(* PLC project CoDeSys External Library Template, WAGO e!COCKPIT e!COCKPIT, author 3S - Smart Software Solutions GmbH *)
(* stored: creationDateTime 2019-10-29T12:37:19.7309586, version 3.5.5.30, modificationDateTime 2019-10-29T12:36:39.3744516, organization 3S - Smart Software Solutions GmbH *)
(* Library project template with all possible element types, docu and a sample project structure *)

FUNCTION_BLOCK fbPPPSZadajnikSR04P
  VAR_INPUT
    sKomunikat : alSTRINGKomunikat;  (* komunikat z systemu zewnętrznego *)
    intTablicaKomunikatowRozmiar : INT;  (* rozmiar tablicy danych wysyłkowych *)
    intModbusOdczytZapisZadanieRozmiar : INT;  (* rozmiar tablicy danych modbusa *)
    xTablicaKomunikatowHold : BOOL;  (* wstrzymanie komunikacji mniej ważnych komunikatów *)
    sIdInstancji : STRING;  (* parametr ID rolety np NS02L*202IBM**** *)
    sIdAplikacji : STRING;  (* parametr ID aplikacji np SO*******ECL*000 *)
    sMnemonik : STRING;  (* mnemonik właściciela - BCB* *)
    sMACAdres : STRING;  (* MAC adres sterownika *)
    sDaneZapasowe : STRING;  (* 6 znaków zapasu *)
    tCzasOpoznieniaRestartu : TIME;  (* czas opóźnienia po którym zaczynają być raportowane wartości *)
    sTypPomieszczenia : STRING;  (* typ pomieszczenia *)
    bAdres : BYTE;
    bKanalEnOcean : BYTE;
    sEnOceanID : STRING(10);
    tMinimalnyCzasRaportowania : TIME;
    tMaksymalnyCzasRaportowania : TIME;
    tCzasTimeoutEnOcean : TIME;
    xAutonomizacja : BOOL;
    xAutonomizacjaSztuczna : BOOL;
    xGlobalnaAutomatycznaKonfiguracja : BOOL;
    tCzestotliwoscAutomatycznejKonfiguracji : TIME;
    rRegulatorTemperaturyKp : REAL;
    rRegulatorTemperaturyTi : REAL;
    rRegulatorTemperaturyDeadZone : REAL;
    rTrybPracyAutonomizacja : REAL;  (* Domyślny tryb pracy *)
    rTemperaturaBazowaAutoAutonomizacja : REAL;  (* Domyślna wartość nastawy temperatury bazowej w trybie automatycznym *)
    rTemperaturaBazowaManAutonomizacja : REAL;  (* Domyślna wartość nastawy temperatury bazowej w trybie manualnym *)
    rSkalaPotencjometruAutonomizacja : REAL;  (* Domyślna skala potencjomentru *)
    rTemperaturaBazowaHMI : REAL := 293.15;  (* Temperatura bazowa z HMI *)
    intTrybPracyHMI : INT := 1;  (* 0 - ręczny; 1 - auto *)
    xPokazPanelHMI : BOOL := TRUE;  (* 0 - widoczny; 1 - niewidoczny *)
  END_VAR
  VAR_IN_OUT
    arModbusOdczytCykliczny : ARRAY[1..5000] OF typModbusOdczytCykliczny;
    arModbusStatusKomunikacji : ARRAY[1..256] OF INT;
    arModbusOdczytZapisZadanie : ARRAY[1..1000] OF typModbusOdczytZapisZadanie;
    intModbusOdczytZapisZadanieZnacznikZapisu : INT;
    arTablicaKomunikatow : alARRAYTablicaKomunikatow;
    intTablicaKomunikatowZnacznikZapisu : INT;
  END_VAR
  VAR_OUTPUT
    rWyjscieRgulatoraTemperatury : REAL;
    rDiagnostykaTemperaturaPomieszczenia : REAL;
    rDiagnostykaTemperaturaNastawiona : REAL;
    rDiagnostykaTemperaturaBazowa : REAL;
    rDiagnostykaKorektaTemperaturyPotencjometru : REAL;
    rDiagnostykaWyjscieRgulatoraTemperatury : REAL;
    intDiagnostykaTrybPracy : INT;
    sDiagnostykaEnOceanIDodczytany : STRING(10);
    wDiagnostykaCzasOdOstatniegoKomunikatu : WORD;
    rTemperaturaPomieszczenia : REAL;
  END_VAR
  VAR CONSTANT
    uintLiczbaRejestrowNaKanal : UINT := 20;
    uintPierwszyRejestr : UINT := 200;
    wEnOceanFunction : WORD := 16;
    wEnOceanType : WORD := 3;
    wEnOceanManufacturer : WORD := 2;
    intDomyslneHarmonogram : INT := enumPPPSHarmonogramy.Komfort;  (* domyślne nastawy po restarcie sterownika *)
    rDomyslneTemperaturaBazowaKomfort : REAL := 293.15;
    rDomyslneTemperaturaBazowaEkonomiczny : REAL := 292.15;
  END_VAR
  VAR
    uintFunctionModbusAdres : UINT;  (* definicja adresów rejestrów modbusowych *)
    uintTypeModbusAdres : UINT;
    uintManufacturerModbusAdres : UINT;
    uintEnOceanIDHiModbusAdres : UINT;
    uintEnOceanIDLoModbusAdres : UINT;
    uintCzasOdOstatniegoKomunikatuModbusAdres : UINT;
    uintPustyRejestr1ModbusAdres : UINT;
    uintStatusUrzadzeniaModbusAdres : UINT;
    uintPustyRejestr2ModbusAdres : UINT;
    uintTemperaturaPomieszczeniaOdczytanaModbusAdres : UINT;
    uintNastawaPotencjometruModbusAdres : UINT;
    xPierwszySkan : BOOL := TRUE;  (* uintLiczbaTelegramowModbusAdres : UINT; zmienne operacyjne *)
    intPetlaPierwszySkan : INT := 1;
    intRozkazTymczasowy : INT;
    arNastawyRegulatoraTemperatury : typConfigPIDController;
    fbRegulatorTemperatury : FbPIDController;
    intBlokadaWykonywaniaRozkazow : INT;
    intBlokadaWykonywaniaRozkazowZaraportowana : INT;
    intTrybPracy : INT;  (* Tryb pracy regulatora. *)
    intTrybPracyZaraportowana : INT;
    xTrybPracyZapisz : BOOL;  (* Trigger zapisu wartości w pamięci urządzenia. *)
    rTrybPracyZapis : REAL;  (* Wartość do zapisania w pamięci urządzenia. *)
    rTemperaturaBazowaAuto : REAL := 293.15;  (* Temperatura bazowa trybu automatycznego. *)
    rTemperaturaBazowaAutoZaraportowana : REAL;
    xTemperaturaBazowaAutoZapisz : BOOL;  (* Trigger zapisu wartości w pamięci urządzenia. *)
    rTemperaturaBazowaAutoZapis : REAL;  (* Wartość do zapisania w pamięci urządzenia. *)
    rTemperaturaBazowaMan : REAL := 293.15;  (* Temperatura bazowa trybu manualnego. *)
    rTemperaturaBazowaManZaraportowana : REAL;
    xTemperaturaBazowaManZapisz : BOOL;  (* Trigger zapisu wartości w pamięci urządzenia. *)
    rTemperaturaBazowaManZapis : REAL;  (* Wartość do zapisania w pamięci urządzenia. *)
    rSkalaPotencjometru : REAL;  (* Skala Potencjometru *)
    rSkalaPotencjometruZaraportowana : REAL;
    xSkalaPotencjometruZapisz : BOOL;  (* Trigger zapisu wartości w pamięci urządzenia. *)
    rSkalaPotencjometruZapis : REAL;  (* Wartość do zapisania w pamięci urządzenia. *)
    fbZadanieGrzania : fbFiltrWartoscAnalogowa;
    rZadanieGrzania : REAL;  (* Zadana grzania *)
    fbZadanieGrzaniaRaport : fbFiltrWartoscAnalogowa;
    rZadanieGrzaniaRaport : REAL;  (* Zadana grzania (raportowana) *)
    rZadanieGrzaniaRaportZaraportowana : REAL;
    rWartoscWejsciowaTemperaturyNastawionej : REAL;
    fbWyslanieKonfiguracji : TON;  (* definicja zmiennych i FB do odczytu wartości z modbusa *)
    xPozwolenieNaAutomatycznaKonfiguracje : BOOL;
    xResetTimerautomatycznejKonfiguracji : BOOL;
    wFunctionEnOceanOdczytana : WORD;
    wTypeEnOceanOdczytana : WORD;
    wManufacturerEnOceanOdczytana : WORD;
    sEnOceanIDodczytany : STRING(10);
    wEnOceanIDHi : WORD;
    wEnOceanIDLo : WORD;
    wEnOceanIDHiZapis : WORD;
    wEnOceanIDLoZapis : WORD;
    wCzasOdOstatniegoKomunikatu : WORD;
    fbTimeoutEnOcean : TON;
    wStatusUrzadzenia : WORD;
    wLiczbaTelegramow : WORD;
    uintLiczbaTelegramow : UINT;
    wPustyRejestr1 : WORD;  (* Rejestry odczytywane dla zgrupowania zapytania rejestrów Modbus *)
    wPustyRejestr2 : WORD;
    wTemperaturaPomieszczeniaOdczytana : WORD;
    fbTemperaturaPomieszczenia : fbFiltrWartoscAnalogowa;
    rTemperaturaPomieszczeniaZaraportowana : REAL;
    wNastawaPotencjometru : WORD;
    rTemperaturaNastawiona : REAL;
    rTemperaturaNastawionaZaraportowana : REAL;
    xPoInicjalizacji : BOOL := FALSE;  (* inicjalizacja *)
    fbInicjalizacyjnyTimer : TON;
    sDane : alSTRINGKomunikat;
    sWyslanyKomunikat : alSTRINGKomunikat;
    sKomunikatPamiec : alSTRINGKomunikat;
    sWyslanyKomunikatDummy : alSTRINGKomunikat;
    intPetla : INT;
    arErrorStan : ARRAY[0..3] OF INT;  (* tablica przechowująca statusy alarmowe *)
    arErrorKlasa : ARRAY[0..3] OF INT;  (* tablica przechowująca klasy danych alarmów *)
    sTempWartoscAtrybutu : STRING;
    rTempWartoscAtrybutu : REAL;
    intTempWartoscAtrybutu : INT;
    xRaport : BOOL;
    uintFunctionAdres : UINT;
    sPlakietkaHMI : STRING;  (* Plakietka pomieszczenia zawierająca numer piętra i pomieszczenia (na potrzeby webvisu) *)
    fnPrzywrocDomyslne : R_TRIG;  (* Przywracanie domyślnych wartości nastaw *)
    fbTaktowanieZapisywaniaModbus : TON;  (* Cykliczne żądanie zapisu danych do urządzenia *)
    xBrakKomunikacjiEnOcean : BOOL;  (* Brak komunikacji z urządzeniem po enOcean *)
    tonBrakKomunikacjiPLC : TON;
    xBrakKomunikacjiPLC : BOOL;
    xBrakKomunikacjiIZE : BOOL;
    rTemperaturaPomieszczeniaPamiec : REAL;  (* Temperatura zapamiętana w celu porównania z aktualną *)
    xBrakZmianyTemperatury : BOOL;  (* Flaga braku zmiany temperatury *)
    fbBrakZmianyTemperaturyTimer : TON;  (* Timer braku zmiany temperatury (24 godziny) *)
    xBladBrakZmianyTemperatury : BOOL;  (* Błąd braku zmiany temperatury *)
    xOsiagniecieTemperaturyZadanej : BOOL := FALSE;  (* Sprawdzanie czy została osiągnęta zadana temperatura *)
    xOsiagniecieTemperaturyZadanejZaraportowana : BOOL := FALSE;
    xFlagaTrybuPracy : BOOL := FALSE;
    rRoznicaTemperaturyZadanejOrazZaraportowanej : REAL;
  END_VAR

            (*			
Autor:					Paweł Kąkol, 2018-08-06, Artur Wyszomirski
Prawa majątkowe: 		Solwena Sp. z o.o., 
Aktualizacje:			
						2018-08-27-PK: dodanie algorytmu nadpisywania konfiguracji (uczenia) anteny
						2018-09-10-PK: dodanie regulatora temperatury oraz obsługi atrybutów potrzebnych do zadajnika z regulatorem, dodanie alarmowania Timeout komunikacji EnOcean
						2018-09-24-AWy: obsługa trybu manualnego i automatycznego
						2018-09-25-PK: dodanie domyślnego przyjmowania 21 st. C po restarcie sterownika, zanim nastąpi Autonomizacja i komunikacja z IZE.
						2018-15-10-AWy: obsługa harmonogramów
						2018-23-10-JB: przygotowanie atrybutów i alarmów do komunikacji z IZE
						2018-12-12-JB: napisanie od nowa obsługi ramek typu C i Q
						2019-02-26-JB: zmiana deadbandów w filtrach analogowych
						2019-04-08-AWy: usunięcie buga braku wysterowania grzejników w trybie manualnym (usunięcie intTrybPracy <> enumPPPSZadajnikTrybPracy.Manualny AND z linii 473)
						2019-05-13-AWy: zmiana wartości umieszczonej w atrybucie STERGRZ. Wartość rZadanieGrzania jest dzielona przez 100 tak, aby zakres STERGRZ mieścił się między 0 a 1.
						2019-05-16-AWy: modyfikacja warunku na raportowanie. Dopisane: AND arModbusStatusKomunikacji[bAdres] = enumModbusStatus.KomunikacjaPrawidlowa AND xPoInicjalizacji 
						2019-05-17-AWy: rozbicie zmiennej rTemperaturaBazowa na rTemperaturaBazowaAuto i rTemperaturaBazowaMan
						2019-05-21-AWy: modyfikacja przepisywania temperatury bazowej z IZE do lokalnej podczas regulacji IZE. 
						2019-06-05-AWy: załadowanie domyślnych trybów pracy i nastaw po przejściu w tryb autonomizacji
						2019-08-05-AWy: dodanie zmiennej sPlakietkaHMI.
						2019-08-14-AWy: zmiana fbPrzywrocDomyslne z przerzutnika RS na R_TRIG.
						2019-09-23-AWy: modyfikacja generowania wartości zmiennej xBrakKomunikacjiPLC
						2019-10-09-AWy: uzależnienie wystąpienia alarmu braku zmiany temperatury od stanu komunikacji 
						2019-10-10-AWy: przywrócenie zmiennej xBrakKomunikacjiEnOcean na potrzeby alarmów i webvisu z I etapu ENGIE
						2019-10-21-AWy: dodanie dodatkowego filtrowania zadanej grzania przy wysyłaniu ramek do IZE
						2019-10-22-AWy: usunięcie uintLiczbaTelegramowModbusAdres z odczytu po Modbusie
						
Opis:					fb służy do komunikacji po Modbus RTU za pośrednictwem bramek (STC65-RS485) EnOcean z zadajnikami FCP0 (SR04P) na budynkach PPP Sopot (ENGIE) 
*)

// Inicjalizacja sterownika
fbInicjalizacyjnyTimer(IN := NOT xPoInicjalizacji , PT := tCzasOpoznieniaRestartu);
IF fbInicjalizacyjnyTimer.Q THEN
	intTrybPracyZaraportowana := intTrybPracy;
	rTemperaturaBazowaAutoZaraportowana := rTemperaturaBazowaAuto;
	rTemperaturaBazowaManZaraportowana := rTemperaturaBazowaMan;
	rSkalaPotencjometruZaraportowana := rSkalaPotencjometru;
	rTemperaturaNastawionaZaraportowana := rTemperaturaNastawiona;
	rTemperaturaPomieszczeniaZaraportowana := rTemperaturaPomieszczenia;
	rZadanieGrzaniaRaportZaraportowana := rZadanieGrzaniaRaport;
	xOsiagniecieTemperaturyZadanej := xOsiagniecieTemperaturyZadanejZaraportowana;
	xPoInicjalizacji := TRUE;
END_IF

// Włącz autonomizację jeśli sterownik jest w stanie inicjalizacji lub nastąpiło wymuszenie autonomizacji
IF NOT xPoInicjalizacji OR xAutonomizacjaSztuczna = TRUE THEN
	xAutonomizacja := TRUE;
END_IF 

// Kontrola komunikacji
tonBrakKomunikacjiPLC(IN := (wCzasOdOstatniegoKomunikatu > 180 OR arModbusStatusKomunikacji[bAdres] <> enumModbusStatus.KomunikacjaPrawidlowa), PT := T#180S);
IF tonBrakKomunikacjiPLC.Q THEN
	xBrakKomunikacjiPLC := TRUE;
ELSE
	xBrakKomunikacjiPLC := FALSE;
END_IF

IF xAutonomizacja THEN
	xBrakKomunikacjiIZE := TRUE;
ELSE
	xBrakKomunikacjiIZE := FALSE;
END_IF

IF xPierwszySkan THEN
	xPierwszySkan := FALSE;
	WHILE arModbusOdczytCykliczny[intPetlaPierwszySkan].bAdresUrzadzenia <> 0 DO
		intPetlaPierwszySkan := intPetlaPierwszySkan + 1;
	END_WHILE
	
	//ustawienie parametrów regulatora temperatury
	arNastawyRegulatoraTemperatury.rKp := rRegulatorTemperaturyKp;
	arNastawyRegulatoraTemperatury.rTn := rRegulatorTemperaturyTi;
	arNastawyRegulatoraTemperatury.rTd := 0.0;
	arNastawyRegulatoraTemperatury.rOutputMax := 100.0;
	arNastawyRegulatoraTemperatury.rOutputMin := 0.0;
	arNastawyRegulatoraTemperatury.xPresetOn := TRUE;
	arNastawyRegulatoraTemperatury.rPresetValueOn := 0.0;
	arNastawyRegulatoraTemperatury.rPresetValueOff := 0.0;
	arNastawyRegulatoraTemperatury.rDeadZone := rRegulatorTemperaturyDeadZone;
	
	//wyznaczenie adresów rejestrów modbusowych
	uintFunctionModbusAdres := uintPierwszyRejestr + (uintLiczbaRejestrowNaKanal * (BYTE_TO_UINT(bKanalEnOcean) - 1));
	uintTypeModbusAdres := uintFunctionModbusAdres + 1;
	uintManufacturerModbusAdres := uintFunctionModbusAdres + 2;
	
	uintEnOceanIDHiModbusAdres := uintFunctionModbusAdres + 3;
	uintEnOceanIDLoModbusAdres := uintFunctionModbusAdres + 4;
	uintCzasOdOstatniegoKomunikatuModbusAdres := uintFunctionModbusAdres + 6;
	uintPustyRejestr1ModbusAdres := uintFunctionModbusAdres + 7;
	uintStatusUrzadzeniaModbusAdres := uintFunctionModbusAdres + 8;
	uintPustyRejestr2ModbusAdres := uintFunctionModbusAdres + 9;
	uintTemperaturaPomieszczeniaOdczytanaModbusAdres := uintFunctionModbusAdres + 10;
	uintNastawaPotencjometruModbusAdres := uintFunctionModbusAdres + 11;
	//uintLiczbaTelegramowModbusAdres := uintFunctionModbusAdres + 19;
	
//deklaracja rejestrow do odczytu
	//rejestry
	arModbusOdczytCykliczny[intPetlaPierwszySkan].bAdresUrzadzenia := bAdres;
	arModbusOdczytCykliczny[intPetlaPierwszySkan].bFunkcja := TO_BYTE(enumModbusKodyFunkcji.OdczytNRejestrow);
	arModbusOdczytCykliczny[intPetlaPierwszySkan].uiAdresRejestru := uintFunctionModbusAdres;
	arModbusOdczytCykliczny[intPetlaPierwszySkan].ltCzestotliwosc := TIME_TO_LTIME(tMaksymalnyCzasRaportowania);
	arModbusOdczytCykliczny[intPetlaPierwszySkan].pZmiennaReferencyjna := ADR(wFunctionEnOceanOdczytana);
	intPetlaPierwszySkan := intPetlaPierwszySkan + 1;
	
	arModbusOdczytCykliczny[intPetlaPierwszySkan].bAdresUrzadzenia := bAdres;
	arModbusOdczytCykliczny[intPetlaPierwszySkan].bFunkcja := TO_BYTE(enumModbusKodyFunkcji.OdczytNRejestrow);
	arModbusOdczytCykliczny[intPetlaPierwszySkan].uiAdresRejestru := uintTypeModbusAdres;
	arModbusOdczytCykliczny[intPetlaPierwszySkan].ltCzestotliwosc := TIME_TO_LTIME(tMaksymalnyCzasRaportowania);
	arModbusOdczytCykliczny[intPetlaPierwszySkan].pZmiennaReferencyjna := ADR(wTypeEnOceanOdczytana);
	intPetlaPierwszySkan := intPetlaPierwszySkan + 1;
	
	arModbusOdczytCykliczny[intPetlaPierwszySkan].bAdresUrzadzenia := bAdres;
	arModbusOdczytCykliczny[intPetlaPierwszySkan].bFunkcja := TO_BYTE(enumModbusKodyFunkcji.OdczytNRejestrow);
	arModbusOdczytCykliczny[intPetlaPierwszySkan].uiAdresRejestru := uintManufacturerModbusAdres;
	arModbusOdczytCykliczny[intPetlaPierwszySkan].ltCzestotliwosc := TIME_TO_LTIME(tMaksymalnyCzasRaportowania);
	arModbusOdczytCykliczny[intPetlaPierwszySkan].pZmiennaReferencyjna := ADR(wManufacturerEnOceanOdczytana);
	intPetlaPierwszySkan := intPetlaPierwszySkan + 1;
	
	arModbusOdczytCykliczny[intPetlaPierwszySkan].bAdresUrzadzenia := bAdres;
	arModbusOdczytCykliczny[intPetlaPierwszySkan].bFunkcja := TO_BYTE(enumModbusKodyFunkcji.OdczytNRejestrow);
	arModbusOdczytCykliczny[intPetlaPierwszySkan].uiAdresRejestru := uintEnOceanIDHiModbusAdres;
	arModbusOdczytCykliczny[intPetlaPierwszySkan].ltCzestotliwosc := TIME_TO_LTIME(tMaksymalnyCzasRaportowania);
	arModbusOdczytCykliczny[intPetlaPierwszySkan].pZmiennaReferencyjna := ADR(wEnOceanIDHi);
	intPetlaPierwszySkan := intPetlaPierwszySkan + 1;
	
	arModbusOdczytCykliczny[intPetlaPierwszySkan].bAdresUrzadzenia := bAdres;
	arModbusOdczytCykliczny[intPetlaPierwszySkan].bFunkcja := TO_BYTE(enumModbusKodyFunkcji.OdczytNRejestrow);
	arModbusOdczytCykliczny[intPetlaPierwszySkan].uiAdresRejestru := uintEnOceanIDLoModbusAdres;
	arModbusOdczytCykliczny[intPetlaPierwszySkan].ltCzestotliwosc := TIME_TO_LTIME(tMaksymalnyCzasRaportowania);
	arModbusOdczytCykliczny[intPetlaPierwszySkan].pZmiennaReferencyjna := ADR(wEnOceanIDLo);
	intPetlaPierwszySkan := intPetlaPierwszySkan + 1;
	
	arModbusOdczytCykliczny[intPetlaPierwszySkan].bAdresUrzadzenia := bAdres;
	arModbusOdczytCykliczny[intPetlaPierwszySkan].bFunkcja := TO_BYTE(enumModbusKodyFunkcji.OdczytNRejestrow);
	arModbusOdczytCykliczny[intPetlaPierwszySkan].uiAdresRejestru := uintCzasOdOstatniegoKomunikatuModbusAdres;
	arModbusOdczytCykliczny[intPetlaPierwszySkan].ltCzestotliwosc := TIME_TO_LTIME(tMinimalnyCzasRaportowania);
	arModbusOdczytCykliczny[intPetlaPierwszySkan].pZmiennaReferencyjna := ADR(wCzasOdOstatniegoKomunikatu);
	intPetlaPierwszySkan := intPetlaPierwszySkan + 1;
	
	arModbusOdczytCykliczny[intPetlaPierwszySkan].bAdresUrzadzenia := bAdres;
	arModbusOdczytCykliczny[intPetlaPierwszySkan].bFunkcja := TO_BYTE(enumModbusKodyFunkcji.OdczytNRejestrow);
	arModbusOdczytCykliczny[intPetlaPierwszySkan].uiAdresRejestru := uintPustyRejestr1ModbusAdres;
	arModbusOdczytCykliczny[intPetlaPierwszySkan].ltCzestotliwosc := TIME_TO_LTIME(tMinimalnyCzasRaportowania);
	arModbusOdczytCykliczny[intPetlaPierwszySkan].pZmiennaReferencyjna := ADR(wPustyRejestr1);
	intPetlaPierwszySkan := intPetlaPierwszySkan + 1;
	
	arModbusOdczytCykliczny[intPetlaPierwszySkan].bAdresUrzadzenia := bAdres;
	arModbusOdczytCykliczny[intPetlaPierwszySkan].bFunkcja := TO_BYTE(enumModbusKodyFunkcji.OdczytNRejestrow);
	arModbusOdczytCykliczny[intPetlaPierwszySkan].uiAdresRejestru := uintStatusUrzadzeniaModbusAdres;
	arModbusOdczytCykliczny[intPetlaPierwszySkan].ltCzestotliwosc := TIME_TO_LTIME(tMinimalnyCzasRaportowania);
	arModbusOdczytCykliczny[intPetlaPierwszySkan].pZmiennaReferencyjna := ADR(wStatusUrzadzenia);
	intPetlaPierwszySkan := intPetlaPierwszySkan + 1;
	
	arModbusOdczytCykliczny[intPetlaPierwszySkan].bAdresUrzadzenia := bAdres;
	arModbusOdczytCykliczny[intPetlaPierwszySkan].bFunkcja := TO_BYTE(enumModbusKodyFunkcji.OdczytNRejestrow);
	arModbusOdczytCykliczny[intPetlaPierwszySkan].uiAdresRejestru := uintPustyRejestr2ModbusAdres;
	arModbusOdczytCykliczny[intPetlaPierwszySkan].ltCzestotliwosc := TIME_TO_LTIME(tMinimalnyCzasRaportowania);
	arModbusOdczytCykliczny[intPetlaPierwszySkan].pZmiennaReferencyjna := ADR(wPustyRejestr2);
	intPetlaPierwszySkan := intPetlaPierwszySkan + 1;
	
	arModbusOdczytCykliczny[intPetlaPierwszySkan].bAdresUrzadzenia := bAdres;
	arModbusOdczytCykliczny[intPetlaPierwszySkan].bFunkcja := TO_BYTE(enumModbusKodyFunkcji.OdczytNRejestrow);
	arModbusOdczytCykliczny[intPetlaPierwszySkan].uiAdresRejestru := uintTemperaturaPomieszczeniaOdczytanaModbusAdres;
	arModbusOdczytCykliczny[intPetlaPierwszySkan].ltCzestotliwosc := TIME_TO_LTIME(tMinimalnyCzasRaportowania);
	arModbusOdczytCykliczny[intPetlaPierwszySkan].pZmiennaReferencyjna := ADR(wTemperaturaPomieszczeniaOdczytana);
	intPetlaPierwszySkan := intPetlaPierwszySkan + 1;	
	
	arModbusOdczytCykliczny[intPetlaPierwszySkan].bAdresUrzadzenia := bAdres;
	arModbusOdczytCykliczny[intPetlaPierwszySkan].bFunkcja := TO_BYTE(enumModbusKodyFunkcji.OdczytNRejestrow);
	arModbusOdczytCykliczny[intPetlaPierwszySkan].uiAdresRejestru := uintNastawaPotencjometruModbusAdres;
	arModbusOdczytCykliczny[intPetlaPierwszySkan].ltCzestotliwosc := TIME_TO_LTIME(tMinimalnyCzasRaportowania);
	arModbusOdczytCykliczny[intPetlaPierwszySkan].pZmiennaReferencyjna := ADR(wNastawaPotencjometru);
	intPetlaPierwszySkan := intPetlaPierwszySkan + 1;
(*	
	arModbusOdczytCykliczny[intPetlaPierwszySkan].bAdresUrzadzenia := bAdres;
	arModbusOdczytCykliczny[intPetlaPierwszySkan].bFunkcja := TO_BYTE(enumModbusKodyFunkcji.OdczytNRejestrow);
	arModbusOdczytCykliczny[intPetlaPierwszySkan].uiAdresRejestru := uintLiczbaTelegramowModbusAdres;
	arModbusOdczytCykliczny[intPetlaPierwszySkan].ltCzestotliwosc := TIME_TO_LTIME(tMinimalnyCzasRaportowania);
	arModbusOdczytCykliczny[intPetlaPierwszySkan].pZmiennaReferencyjna := ADR(wLiczbaTelegramow);
	intPetlaPierwszySkan := intPetlaPierwszySkan + 1;
*)	
(*	//przyjęcie nastaw domyślnych do momentu uzyskania nastaw z IZE lub przejścia w autonomizację
	IF intDomyslneHarmonogram = enumPPPSHarmonogramy.Ekonomiczny THEN
		rTemperaturaBazowaAuto := rDomyslneTemperaturaBazowaEkonomiczny;
	ELSE
		rTemperaturaBazowaAuto := rDomyslneTemperaturaBazowaKomfort;													
	END_IF
	intTrybPracy := enumPPPSZadajnikTrybPracy.Automatyczny;
	rSkalaPotencjometru := rSkalaPotencjometruAutonomizacja;	*)
END_IF

// Obsługa komunikatu przychodzacego z IZE
IF 	sKomunikat <> sKomunikatPamiec AND xPoInicjalizacji THEN
	sKomunikatPamiec := sKomunikat;
	IF fnIDOdbiorcyMatch(sKomunikat , sIdInstancji) THEN
		sDane := '';
		// Rozkaz typu C
		IF fnKomunikatTyp(sKomunikat) = 'C' AND NOT xAutonomizacja THEN
			// Blokada wykonywania rozkazów
			IF fnKomunikatDaneSzukajWartosci(sKomunikat,'BLOK=') = '0' THEN
				IF intBlokadaWykonywaniaRozkazow = 1 THEN
					intBlokadaWykonywaniaRozkazow := 0;
					xRaport := TRUE;
					ELSE	
					IF sDane <> '' THEN
					sDane := CONCAT(sDane , ';');
					END_IF
					sDane := CONCAT(sDane , 'BLOK=0');
				END_IF
			END_IF
			IF fnKomunikatDaneSzukajWartosci(sKomunikat,'BLOK=') = '1' THEN
				IF intBlokadaWykonywaniaRozkazow = 0 THEN
					intBlokadaWykonywaniaRozkazow := 1;
					xRaport := TRUE;
					ELSE
					IF sDane <> '' THEN
					sDane := CONCAT(sDane , ';');
					END_IF					
					sDane := CONCAT(sDane , 'BLOK=1');
				END_IF
			END_IF		

			IF intBlokadaWykonywaniaRozkazow = 0 THEN
				// Tryby pracy 
				fnKomunikatDaneZnajdzPorownajZapisz(sKomunikat := sKomunikat,
					sAtrybut := 'TRYB=',
					rAtrybutWartosc := rTrybPracyZapis,
					sDane := sDane,
					xAtrybutZapisz => xTrybPracyZapisz);	
				// Temperatura bazowa w trybie automatycznym
				fnKomunikatDaneZnajdzPorownajZapisz(sKomunikat := sKomunikat,
					sAtrybut := 'TEMPBAZAUTO=',
					rAtrybutWartosc := rTemperaturaBazowaAutoZapis,
					sDane := sDane,
					xAtrybutZapisz => xTemperaturaBazowaAutoZapisz);	
				// Temperatura bazowa w trybie manualnym
				fnKomunikatDaneZnajdzPorownajZapisz(sKomunikat := sKomunikat,
					sAtrybut := 'TEMPBAZMAN=',
					rAtrybutWartosc := rTemperaturaBazowaManZapis,
					sDane := sDane,
					xAtrybutZapisz => xTemperaturaBazowaManZapisz);
				// Skala potencjometru
				fnKomunikatDaneZnajdzPorownajZapisz(sKomunikat := sKomunikat,
					sAtrybut := 'SKALAPOT=',
					rAtrybutWartosc := rSkalaPotencjometruZapis,
					sDane := sDane,
					xAtrybutZapisz => xSkalaPotencjometruZapisz);
			END_IF
		END_IF	

		// Zapytanie typu Q
		IF fnKomunikatTyp(sKomunikat) = 'Q' AND arModbusStatusKomunikacji[bAdres] = enumModbusStatus.KomunikacjaPrawidlowa THEN
			IF fnKomunikatDaneSzukajWartosci(sKomunikat , 'BLOK=') = '?' OR fnKomunikatDaneSzukajWartosci(sKomunikat , 'ALL=') = '?' THEN
				fnKomunikatDaneDodaj(sDane := sDane , sAtrybut := 'BLOK=' , sWartosc := INT_TO_STRING(intBlokadaWykonywaniaRozkazow));	
			END_IF
			IF fnKomunikatDaneSzukajWartosci(sKomunikat , 'TRYB=') = '?' OR fnKomunikatDaneSzukajWartosci(sKomunikat , 'ALL=') = '?' THEN
				fnKomunikatDaneDodaj(sDane := sDane , sAtrybut := 'TRYB=' , sWartosc := INT_TO_STRING(intTrybPracy));	
			END_IF
			IF (fnKomunikatDaneSzukajWartosci(sKomunikat , 'TEMPBAZMAN=') = '?' OR fnKomunikatDaneSzukajWartosci(sKomunikat , 'ALL=') = '?') THEN
				fnKomunikatDaneDodaj(sDane := sDane , sAtrybut := 'TEMPBAZMAN=' , sWartosc := REAL_TO_STRING(rTemperaturaBazowaMan));	
			END_IF
			IF (fnKomunikatDaneSzukajWartosci(sKomunikat , 'TEMPBAZAUTO=') = '?' OR fnKomunikatDaneSzukajWartosci(sKomunikat , 'ALL=') = '?') THEN
				fnKomunikatDaneDodaj(sDane := sDane , sAtrybut := 'TEMPBAZAUTO=' , sWartosc := REAL_TO_STRING(rTemperaturaBazowaAuto));	
			END_IF
			IF fnKomunikatDaneSzukajWartosci(sKomunikat , 'SKALAPOT=') = '?' OR fnKomunikatDaneSzukajWartosci(sKomunikat , 'ALL=') = '?' THEN
				fnKomunikatDaneDodaj(sDane := sDane , sAtrybut := 'SKALAPOT=' , sWartosc := REAL_TO_STRING(rSkalaPotencjometru));	
			END_IF
			IF fnKomunikatDaneSzukajWartosci(sKomunikat , 'TEMP=') = '?' OR fnKomunikatDaneSzukajWartosci(sKomunikat , 'ALL=') = '?' THEN
				fnKomunikatDaneDodaj(sDane := sDane , sAtrybut := 'TEMP=' , sWartosc := REAL_TO_STRING(rTemperaturaPomieszczenia));	
			END_IF
			IF fnKomunikatDaneSzukajWartosci(sKomunikat , 'STERGRZ=') = '?' OR fnKomunikatDaneSzukajWartosci(sKomunikat , 'ALL=') = '?' THEN
				fnKomunikatDaneDodaj(sDane := sDane , sAtrybut := 'STERGRZ=' , sWartosc := REAL_TO_STRING(rZadanieGrzaniaRaport / 100));	
			END_IF
			IF fnKomunikatDaneSzukajWartosci(sKomunikat , 'TEMPNAS=') = '?' OR fnKomunikatDaneSzukajWartosci(sKomunikat , 'ALL=') = '?' THEN
				fnKomunikatDaneDodaj(sDane := sDane , sAtrybut := 'TEMPNAS=' , sWartosc := REAL_TO_STRING(rTemperaturaNastawiona));	
			END_IF
			IF fnKomunikatDaneSzukajWartosci(sKomunikat , 'DOGRZ=') = '?' OR fnKomunikatDaneSzukajWartosci(sKomunikat , 'ALL=') = '?' THEN
				fnKomunikatDaneDodaj(sDane := sDane , sAtrybut := 'DOGRZ=' , sWartosc := INT_TO_STRING(BOOL_TO_INT(xOsiagniecieTemperaturyZadanej)));	
			END_IF
			//pytanie o stany alarmów
			IF fnKomunikatDaneSzukajWartosci(sKomunikat , 'ALARM=') = '?' OR fnKomunikatDaneSzukajWartosci(sKomunikat , 'ALL=') = '?' THEN
				FOR intPetla := 1 TO 4 BY 1 DO
					//raportowanie typu E (stanów alarmów) na zapytanie typu Q
					IF arErrorStan[intPetla] <> enumAlarmWartosc.StanNieznany THEN
						fnZapiszKomunikat(	sCalyKomunikat := '' ,
											sTypKomunikatu := 'E' ,
											sMnemonik := sMnemonik ,
											sMACAdres := sMACAdres ,
											sIDNadawcy := sIdInstancji ,
											sIDOdbiorcy := sIdAplikacji ,
											sDaneZapasowe := sDaneZapasowe ,
											sDane := fnKomunikatDaneErrorRetry(xAktywny := arErrorStan[intPetla] = enumAlarmWartosc.StanAlarmowy , intKlasa := arErrorKlasa[intPetla] , intNumer := intPetla),
											arTablicaKomunikatow := arTablicaKomunikatow ,
											intTablicaKomunikatowZnacznikZapisu := intTablicaKomunikatowZnacznikZapisu ,
											intTablicaKomunikatowRozmiar := intTablicaKomunikatowRozmiar ,
											sWyslanyKomunikat := sWyslanyKomunikatDummy);
					END_IF
				END_FOR
			END_IF
		END_IF
		
		// Raportowanie typu A
		IF sDane <> '' THEN
			fnZapiszKomunikat(	sCalyKomunikat := '' ,
								sTypKomunikatu := 'A' ,
								sMnemonik := sMnemonik ,
								sMACAdres := sMACAdres ,
								sIDNadawcy := sIdInstancji ,
								sIDOdbiorcy := sIdAplikacji ,
								sDaneZapasowe := sDaneZapasowe ,
								sDane := sDane ,
								arTablicaKomunikatow := arTablicaKomunikatow ,
								intTablicaKomunikatowZnacznikZapisu := intTablicaKomunikatowZnacznikZapisu ,
								intTablicaKomunikatowRozmiar := intTablicaKomunikatowRozmiar ,
								sWyslanyKomunikat := sWyslanyKomunikatDummy);
		END_IF
	END_IF
END_IF

// Przywrócenie wartości domyślnych nastaw krzywej grzewczej i trybów pracy w przypadku restartu sterownika lub przejścia w stan autonomizacji (brak komunikacji z IZE)
fnPrzywrocDomyslne(CLK := xAutonomizacja);
IF fnPrzywrocDomyslne.Q THEN	
	IF intTrybPracy <> REAL_TO_INT(rTrybPracyAutonomizacja) THEN
		rTrybPracyZapis := rTrybPracyAutonomizacja;
		xTrybPracyZapisz := TRUE;
	END_IF
	IF rTemperaturaBazowaAuto <> rTemperaturaBazowaAutoAutonomizacja THEN
		rTemperaturaBazowaAutoZapis := rTemperaturaBazowaAutoAutonomizacja + 273.15;
		xTemperaturaBazowaAutoZapisz := TRUE;
	END_IF
	IF rTemperaturaBazowaMan <> rTemperaturaBazowaManAutonomizacja THEN
		rTemperaturaBazowaManZapis := rTemperaturaBazowaManAutonomizacja;
		xTemperaturaBazowaManZapisz := TRUE;
	END_IF
	IF rSkalaPotencjometru <> rSkalaPotencjometruAutonomizacja THEN
		rSkalaPotencjometruZapis := rSkalaPotencjometruAutonomizacja;
		xSkalaPotencjometruZapisz := TRUE;
	END_IF
END_IF	

// Zapisanie nastaw domyślnych lub otrzymanych w ramce C
IF xTrybPracyZapisz THEN
	intTrybPracy := REAL_TO_INT(rTrybPracyZapis);
	intTrybPracyHMI := REAL_TO_INT(rTrybPracyZapis);
	xTrybPracyZapisz := FALSE;
END_IF
IF xTemperaturaBazowaAutoZapisz THEN
	rTemperaturaBazowaAuto := rTemperaturaBazowaAutoZapis;
	xTemperaturaBazowaAutoZapisz := FALSE;
END_IF
IF xTemperaturaBazowaManZapisz THEN
	rTemperaturaBazowaMan := rTemperaturaBazowaManZapis;
	xTemperaturaBazowaManZapisz := FALSE;
END_IF
IF xSkalaPotencjometruZapisz THEN
	rSkalaPotencjometru := rSkalaPotencjometruZapis;
	xSkalaPotencjometruZapisz := FALSE;
END_IF

// Tryby pracy
IF xAutonomizacja THEN	// W trybie automonizacji pobieraj tryb pracy i temperaturę bazową z panelu WebVisu
	IF intTrybPracyHMI = enumPPPSZadajnikTrybPracy.Manualny THEN	
		intTrybPracy := enumPPPSZadajnikTrybPracy.Manualny;
		rTemperaturaBazowaMan := rTemperaturaBazowaHMI + 273.15;
	ELSE
		intTrybPracy := enumPPPSZadajnikTrybPracy.Automatyczny;
		rTemperaturaBazowaAuto := rTemperaturaBazowaAutoAutonomizacja + 273.15;
	END_IF
ELSE // W trybie sterowania z IZE pobieraj tryb pracy i temperaturę bazową z panelu WebVisu
	IF intTrybPracy = enumPPPSZadajnikTrybPracy.Manualny THEN
		intTrybPracyHMI := enumPPPSZadajnikTrybPracy.Manualny;
		rTemperaturaBazowaHMI := rTemperaturaBazowaMan - 273.15;
	ELSE
		intTrybPracyHMI := enumPPPSZadajnikTrybPracy.Automatyczny;
		rTemperaturaBazowaHMI := rTemperaturaBazowaAuto - 273.15;
	END_IF	
END_IF
						 
IF intTrybPracy = enumPPPSZadajnikTrybPracy.Manualny THEN 	
	rTemperaturaNastawiona := rTemperaturaBazowaMan; // W trybie manualnym nie uwzględniaj nastawy potencjometru na zadajniku
ELSE
	rTemperaturaNastawiona := ((WORD_TO_REAL(wNastawaPotencjometru) - 127.0) * rSkalaPotencjometru / 127.0) + rTemperaturaBazowaAuto; // W trybie automatycznym uwzględnij nastawę Potencjometru
END_IF

//Autokonfiguracja bramki EnOcean
sEnOceanIDodczytany := CONCAT(CONCAT(fnKonwersjaDEC_BYTE_TO_HEX_STRING(INT_TO_BYTE(WORD_TO_INT(wEnOceanIDHi / 256))), fnKonwersjaDEC_BYTE_TO_HEX_STRING(WORD_TO_BYTE(wEnOceanIDHi))), CONCAT(fnKonwersjaDEC_BYTE_TO_HEX_STRING(INT_TO_BYTE(WORD_TO_INT(wEnOceanIDLo / 256))), fnKonwersjaDEC_BYTE_TO_HEX_STRING(WORD_TO_BYTE(wEnOceanIDLo))));

fbWyslanieKonfiguracji(IN := ((xPozwolenieNaAutomatycznaKonfiguracje OR xGlobalnaAutomatycznaKonfiguracja) AND NOT xResetTimerautomatycznejKonfiguracji) , PT := tCzestotliwoscAutomatycznejKonfiguracji);
xResetTimerautomatycznejKonfiguracji := FALSE;

IF((xPozwolenieNaAutomatycznaKonfiguracje OR xGlobalnaAutomatycznaKonfiguracja) AND fbWyslanieKonfiguracji.Q) THEN
	//EnOcean ID urządzenia
	IF sEnOceanID <> sEnOceanIDodczytany THEN
		wEnOceanIDHiZapis := BYTE_TO_WORD(fnKonwersjaHEX_STRING_TO_DEC_BYTE(LEFT(sEnOceanID, 2))) * 256 + BYTE_TO_WORD(fnKonwersjaHEX_STRING_TO_DEC_BYTE(LEFT(RIGHT(sEnOceanID, 6), 2)));
		fnModbusZapisRejestru(	bAdresUrzadzenia := bAdres,
								bFunkcja := INT_TO_BYTE(enumModbusKodyFunkcji.ZapisRejestru),										
								uiAdresRejestru := uintEnOceanIDHiModbusAdres,
								pZmiennaReferencyjna := 0,
								wWartoscDoZapisania := wEnOceanIDHiZapis,
								intModbusOdczytZapisZadanieRozmiar := intModbusOdczytZapisZadanieRozmiar,
								arModbusOdczytZapisZadanie := arModbusOdczytZapisZadanie,
								intModbusOdczytZapisZadanieZnacznikZapisu := intModbusOdczytZapisZadanieZnacznikZapisu);
		wEnOceanIDLoZapis := BYTE_TO_WORD(fnKonwersjaHEX_STRING_TO_DEC_BYTE(LEFT(RIGHT(sEnOceanID, 4), 2))) * 256 + BYTE_TO_WORD(fnKonwersjaHEX_STRING_TO_DEC_BYTE(RIGHT(sEnOceanID, 2)));
		fnModbusZapisRejestru(	bAdresUrzadzenia := bAdres,
								bFunkcja := INT_TO_BYTE(enumModbusKodyFunkcji.ZapisRejestru),										
								uiAdresRejestru := uintEnOceanIDLoModbusAdres,
								pZmiennaReferencyjna := 0,
								wWartoscDoZapisania := wEnOceanIDLoZapis,
								intModbusOdczytZapisZadanieRozmiar := intModbusOdczytZapisZadanieRozmiar,
								arModbusOdczytZapisZadanie := arModbusOdczytZapisZadanie,
								intModbusOdczytZapisZadanieZnacznikZapisu := intModbusOdczytZapisZadanieZnacznikZapisu);
	END_IF
	//stałe wartości dla danego typu urządzeń
	IF wFunctionEnOceanOdczytana <> wEnOceanFunction THEN
		fnModbusZapisRejestru(	bAdresUrzadzenia := bAdres,
								bFunkcja := INT_TO_BYTE(enumModbusKodyFunkcji.ZapisRejestru),										
								uiAdresRejestru := uintFunctionModbusAdres,
								pZmiennaReferencyjna := 0,
								wWartoscDoZapisania := wEnOceanFunction,
								intModbusOdczytZapisZadanieRozmiar := intModbusOdczytZapisZadanieRozmiar,
								arModbusOdczytZapisZadanie := arModbusOdczytZapisZadanie,
								intModbusOdczytZapisZadanieZnacznikZapisu := intModbusOdczytZapisZadanieZnacznikZapisu);
	END_IF
	IF wTypeEnOceanOdczytana <> wEnOceanType THEN
		fnModbusZapisRejestru(	bAdresUrzadzenia := bAdres,
								bFunkcja := INT_TO_BYTE(enumModbusKodyFunkcji.ZapisRejestru),										
								uiAdresRejestru := uintTypeModbusAdres,
								pZmiennaReferencyjna := 0,
								wWartoscDoZapisania := wEnOceanType,
								intModbusOdczytZapisZadanieRozmiar := intModbusOdczytZapisZadanieRozmiar,
								arModbusOdczytZapisZadanie := arModbusOdczytZapisZadanie,
								intModbusOdczytZapisZadanieZnacznikZapisu := intModbusOdczytZapisZadanieZnacznikZapisu);
	END_IF
	IF wManufacturerEnOceanOdczytana <> wEnOceanManufacturer THEN
		fnModbusZapisRejestru(	bAdresUrzadzenia := bAdres,
								bFunkcja := INT_TO_BYTE(enumModbusKodyFunkcji.ZapisRejestru),										
								uiAdresRejestru := uintManufacturerModbusAdres,
								pZmiennaReferencyjna := 0,
								wWartoscDoZapisania := wEnOceanManufacturer,
								intModbusOdczytZapisZadanieRozmiar := intModbusOdczytZapisZadanieRozmiar,
								arModbusOdczytZapisZadanie := arModbusOdczytZapisZadanie,
								intModbusOdczytZapisZadanieZnacznikZapisu := intModbusOdczytZapisZadanieZnacznikZapisu);
	END_IF
	xResetTimerautomatycznejKonfiguracji := TRUE;
END_IF

//sprawdzanie Timeout komunikacji
fbTimeoutEnOcean(IN := ((wCzasOdOstatniegoKomunikatu > 120) AND arModbusStatusKomunikacji[bAdres] = enumModbusStatus.KomunikacjaPrawidlowa) , PT := tCzasTimeoutEnOcean);	
							
fbTemperaturaPomieszczenia(	rWartoscWejsciowa := WORD_TO_REAL(wTemperaturaPomieszczeniaOdczytana),
							rDeadband := 0.1,
							tCzasMinimalny := tMinimalnyCzasRaportowania,
							tCzasMaksymalny := tMaksymalnyCzasRaportowania,
							rWynikMnoznik := (-40.0 / 255.0),
							rWynikOffset := 273.15 + 40.0,
							rWartoscWejsciowaZaraportowana := rTemperaturaPomieszczeniaZaraportowana,
							rWartoscWyjsciowa => rTemperaturaPomieszczenia);

//regulator PI
fbRegulatorTemperatury( xEnable := TRUE,
	rReferenceValue := rTemperaturaNastawiona,
	rActualValue := rTemperaturaPomieszczenia,
	typConfigParameters := arNastawyRegulatoraTemperatury,
	rY => rWyjscieRgulatoraTemperatury);

fbZadanieGrzania(rWartoscWejsciowa := rWyjscieRgulatoraTemperatury,
	rDeadband := 0.25,
	tCzasMinimalny := tMinimalnyCzasRaportowania,
	tCzasMaksymalny := tMaksymalnyCzasRaportowania,
	rWynikMnoznik := 1,
	rWynikOffset := 0.0,
	rWartoscWejsciowaZaraportowana := rZadanieGrzania,
	rWartoscWyjsciowa => rZadanieGrzania);		
	
// Raportowanie zadanej grzania
fbZadanieGrzaniaRaport(rWartoscWejsciowa := rZadanieGrzania,
	rDeadband := 10,
	tCzasMinimalny := tMinimalnyCzasRaportowania,
	tCzasMaksymalny := tMaksymalnyCzasRaportowania,
	rWynikMnoznik := 1,
	rWynikOffset := 0.0,
	rWartoscWejsciowaZaraportowana := rZadanieGrzaniaRaportZaraportowana,
	rWartoscWyjsciowa => rZadanieGrzaniaRaport);		
	
// Nowy filtr "antypyćkowy"
IF rZadanieGrzania < 0.25 THEN
	rZadanieGrzania := 0;
	rZadanieGrzaniaRaport := 0;
ELSIF rZadanieGrzania > 99.75 THEN
	rZadanieGrzania := 100;
	rZadanieGrzaniaRaport := 100;	
END_IF
(*
// FILTR ANTY_PYĆKOWY
rRoznicaTemperaturyZadanejOrazZaraportowanej := rZadanieGrzania - rZadanieGrzaniaZaraportowana;
IF rRoznicaTemperaturyZadanejOrazZaraportowanej < 0.25 AND rRoznicaTemperaturyZadanejOrazZaraportowanej > 0 AND rZadanieGrzania < 1.0 THEN
	rZadanieGrzania := rZadanieGrzaniaZaraportowana;
END_IF	

IF rRoznicaTemperaturyZadanejOrazZaraportowanej > - 0.25 AND rRoznicaTemperaturyZadanejOrazZaraportowanej < 0 AND rZadanieGrzania > 99.0 THEN
	rZadanieGrzania := rZadanieGrzaniaZaraportowana;
END_IF	
	*)		
///////Diagnostyka na czas uruchomień////////
	rDiagnostykaTemperaturaPomieszczenia := rTemperaturaPomieszczenia;
	rDiagnostykaTemperaturaNastawiona := rTemperaturaNastawiona;
	rDiagnostykaTemperaturaBazowa := rTemperaturaBazowaAuto;
	rDiagnostykaKorektaTemperaturyPotencjometru := (WORD_TO_REAL(wNastawaPotencjometru) - 127.0) * rSkalaPotencjometru / 127.0;
	rDiagnostykaWyjscieRgulatoraTemperatury := rWyjscieRgulatoraTemperatury;
	intDiagnostykaTrybPracy := intTrybPracy;
	sDiagnostykaEnOceanIDodczytany := sEnOceanIDodczytany;
	wDiagnostykaCzasOdOstatniegoKomunikatu := wCzasOdOstatniegoKomunikatu;
//////////////////////////////////////////////		
IF (intBlokadaWykonywaniaRozkazow <> intBlokadaWykonywaniaRozkazowZaraportowana OR intTrybPracy <> intTrybPracyZaraportowana OR rTemperaturaBazowaAuto <> rTemperaturaBazowaAutoZaraportowana OR 
	rSkalaPotencjometru <> rSkalaPotencjometruZaraportowana OR rTemperaturaNastawiona <> rTemperaturaNastawionaZaraportowana OR rTemperaturaPomieszczenia <> rTemperaturaPomieszczeniaZaraportowana OR 
	rZadanieGrzaniaRaport <> rZadanieGrzaniaRaportZaraportowana OR xOsiagniecieTemperaturyZadanej <> xOsiagniecieTemperaturyZadanejZaraportowana OR rTemperaturaBazowaMan <> rTemperaturaBazowaManZaraportowana) AND 
	arModbusStatusKomunikacji[bAdres] = enumModbusStatus.KomunikacjaPrawidlowa AND xPoInicjalizacji THEN
	xRaport := TRUE;
END_IF

IF xRaport THEN
	sDane := '';
	xRaport := FALSE;
	IF intBlokadaWykonywaniaRozkazow <> intBlokadaWykonywaniaRozkazowZaraportowana THEN
		intBlokadaWykonywaniaRozkazowZaraportowana := intBlokadaWykonywaniaRozkazow;
		fnKomunikatDaneDodaj(sDane := sDane , sAtrybut := 'BLOK=' , sWartosc := INT_TO_STRING(intBlokadaWykonywaniaRozkazow));	
	END_IF
	IF intTrybPracy <> intTrybPracyZaraportowana THEN
		intTrybPracyZaraportowana := intTrybPracy;
		fnKomunikatDaneDodaj(sDane := sDane , sAtrybut := 'TRYB=' , sWartosc := INT_TO_STRING(intTrybPracy));	
	END_IF
	IF (rTemperaturaBazowaMan <> rTemperaturaBazowaManZaraportowana) THEN
		rTemperaturaBazowaManZaraportowana := rTemperaturaBazowaMan;
		fnKomunikatDaneDodaj(sDane := sDane , sAtrybut := 'TEMPBAZMAN=' , sWartosc := REAL_TO_STRING(rTemperaturaBazowaMan));	
	END_IF
	IF (rTemperaturaBazowaAuto <> rTemperaturaBazowaAutoZaraportowana) THEN
		rTemperaturaBazowaAutoZaraportowana := rTemperaturaBazowaAuto;
		fnKomunikatDaneDodaj(sDane := sDane , sAtrybut := 'TEMPBAZAUTO=' , sWartosc := REAL_TO_STRING(rTemperaturaBazowaAuto));	
	END_IF
	IF rSkalaPotencjometru <> rSkalaPotencjometruZaraportowana THEN
		rSkalaPotencjometruZaraportowana := rSkalaPotencjometru;
		fnKomunikatDaneDodaj(sDane := sDane , sAtrybut := 'SKALAPOT=' , sWartosc := REAL_TO_STRING(rSkalaPotencjometru));	
	END_IF
	IF rTemperaturaNastawiona <> rTemperaturaNastawionaZaraportowana THEN
		rTemperaturaNastawionaZaraportowana := rTemperaturaNastawiona;
		fnKomunikatDaneDodaj(sDane := sDane , sAtrybut := 'TEMPNAS=' , sWartosc := REAL_TO_STRING(rTemperaturaNastawiona));	
	END_IF
	IF rTemperaturaPomieszczenia <> rTemperaturaPomieszczeniaZaraportowana THEN
		rTemperaturaPomieszczeniaZaraportowana := rTemperaturaPomieszczenia;
		fnKomunikatDaneDodaj(sDane := sDane , sAtrybut := 'TEMP=' , sWartosc := REAL_TO_STRING(rTemperaturaPomieszczenia));	
	END_IF
	IF rZadanieGrzaniaRaport <> rZadanieGrzaniaRaportZaraportowana THEN
		rZadanieGrzaniaRaportZaraportowana := rZadanieGrzaniaRaport;	
		fnKomunikatDaneDodaj(sDane := sDane , sAtrybut := 'STERGRZ=' , sWartosc := REAL_TO_STRING(rZadanieGrzaniaRaport / 100));	
	END_IF
	IF xOsiagniecieTemperaturyZadanej <> xOsiagniecieTemperaturyZadanejZaraportowana THEN
		xOsiagniecieTemperaturyZadanejZaraportowana := xOsiagniecieTemperaturyZadanej;
		fnKomunikatDaneDodaj(sDane := sDane , sAtrybut := 'DOGRZ=' , sWartosc := INT_TO_STRING(BOOL_TO_INT(xOsiagniecieTemperaturyZadanej)));	
	END_IF
	
(*	IF rTemperaturaPomieszczeniaMIN <> rTemperaturaPomieszczeniaMINZaraportowana OR rTemperaturaPomieszczeniaMAX <> rTemperaturaPomieszczeniaMAXZaraportowana THEN
		
		fnKomunikatDaneDodaj(sDane := sDane , sAtrybut := 'TEMPPOC=' , sWartosc := REAL_TO_STRING(rTemperaturaPomieszczeniaPOCZATKOWA));
		rTemperaturaPomieszczeniaPOCZATKOWA := rTemperaturaPomieszczenia;
		
		rTemperaturaPomieszczeniaKONCOWA := rTemperaturaPomieszczenia;
		fnKomunikatDaneDodaj(sDane := sDane , sAtrybut := 'TEMPKON=' , sWartosc := REAL_TO_STRING(rTemperaturaPomieszczeniaKONCOWA));
		
		rTemperaturaPomieszczeniaMINZaraportowana := rTemperaturaPomieszczeniaMIN;
		fnKomunikatDaneDodaj(sDane := sDane , sAtrybut := 'TEMPMIN=' , sWartosc := REAL_TO_STRING(rTemperaturaPomieszczeniaMIN));
		rZmiennaProcesowaMinimumTemperatury := 500.0;
		
		rTemperaturaPomieszczeniaMAXZaraportowana := rTemperaturaPomieszczeniaMAX;
		fnKomunikatDaneDodaj(sDane := sDane , sAtrybut := 'TEMPMAX=' , sWartosc := REAL_TO_STRING(rTemperaturaPomieszczeniaMAX));
		rZmiennaProcesowaMaximumTemperatury := -1.0;
		
		fnKomunikatDaneDodaj(sDane := sDane , sAtrybut := 'TEMPSRE=' , sWartosc := REAL_TO_STRING(rTemperaturaPomieszczeniaSREDNIA));
		rTemperaturaPomieszczeniaSREDNIA := 0.0;
		
		fnKomunikatDaneDodaj(sDane := sDane , sAtrybut := 'TEMPMED=' , sWartosc := REAL_TO_STRING(rTemperaturaPomieszczeniaMEDIANA));
		rTemperaturaPomieszczeniaMEDIANA := -1.0;
	END_IF
*)

	IF sDane <> '' AND xPoInicjalizacji THEN
		fnZapiszKomunikat(	sCalyKomunikat := '' ,
							sTypKomunikatu := 'M' ,
							sMnemonik := sMnemonik ,
							sMACAdres := sMACAdres ,
							sIDNadawcy := sIdInstancji ,
							sIDOdbiorcy := sIdAplikacji ,
							sDaneZapasowe := sDaneZapasowe ,
							sDane := sDane ,
							arTablicaKomunikatow := arTablicaKomunikatow ,
							intTablicaKomunikatowZnacznikZapisu := intTablicaKomunikatowZnacznikZapisu ,
							intTablicaKomunikatowRozmiar := intTablicaKomunikatowRozmiar ,
							sWyslanyKomunikat := sWyslanyKomunikat);
	END_IF
END_IF

// Sprawdzanie czy pomiar temperatury działa (odczyt jest niepoprawny, jeśli nie zmienił wartości w przeciągu doby)
IF rTemperaturaPomieszczeniaPamiec = rTemperaturaPomieszczenia THEN
	xBrakZmianyTemperatury := TRUE;
ELSE
	xBrakZmianyTemperatury := FALSE;	
END_IF
fbBrakZmianyTemperaturyTimer(IN := xBrakZmianyTemperatury, PT := T#12H);
rTemperaturaPomieszczeniaPamiec := rTemperaturaPomieszczenia;
IF fbBrakZmianyTemperaturyTimer.Q AND NOT xBrakKomunikacjiPLC THEN
	xBladBrakZmianyTemperatury := TRUE;
ELSE
	xBladBrakZmianyTemperatury := FALSE;
END_IF

// Sprawdzanie czy została osiągnęta zadana temperatura
IF rTemperaturaPomieszczenia >= rTemperaturaNastawiona THEN
	xOsiagniecieTemperaturyZadanej  := TRUE;
END_IF
IF rTemperaturaPomieszczenia <= rTemperaturaNastawiona - 0.4 THEN
	xOsiagniecieTemperaturyZadanej := FALSE;	
END_IF

// obsługa alarmów do zadajnika
	//brak komunikacji po EnOcean
IF arErrorStan[enumPPPSZadajnikError.BrakKomunikacji] <> enumAlarmWartosc.StanAlarmowy AND fbTimeoutEnOcean.Q AND arModbusStatusKomunikacji[bAdres] = enumModbusStatus.KomunikacjaPrawidlowa THEN
	arErrorStan[enumPPPSZadajnikError.BrakKomunikacji] := enumAlarmWartosc.StanAlarmowy;
	xBrakKomunikacjiEnOcean := TRUE;
	arErrorKlasa[enumPPPSZadajnikError.BrakKomunikacji] := enumPPPSZadajnikErrorKlasa.BrakKomunikacji;
	IF xPoInicjalizacji THEN
		fnZapiszKomunikat(	sCalyKomunikat := '' ,
							sTypKomunikatu := 'E' ,
							sMnemonik := sMnemonik ,
							sMACAdres := sMACAdres ,
							sIDNadawcy := sIdInstancji ,
							sIDOdbiorcy := sIdAplikacji ,
							sDaneZapasowe := sDaneZapasowe ,
							sDane := fnKomunikatDaneError(xAktywny := TRUE , intKlasa := enumPPPSZadajnikErrorKlasa.BrakKomunikacji , intNumer := enumPPPSZadajnikError.BrakKomunikacji),
							arTablicaKomunikatow := arTablicaKomunikatow ,
							intTablicaKomunikatowZnacznikZapisu := intTablicaKomunikatowZnacznikZapisu ,
							intTablicaKomunikatowRozmiar := intTablicaKomunikatowRozmiar ,
							sWyslanyKomunikat := sWyslanyKomunikatDummy);
	END_IF
END_IF
IF arErrorStan[enumPPPSZadajnikError.BrakKomunikacji] <> enumAlarmWartosc.StanNormalny AND NOT fbTimeoutEnOcean.Q AND arModbusStatusKomunikacji[bAdres] = enumModbusStatus.KomunikacjaPrawidlowa THEN
	arErrorStan[enumPPPSZadajnikError.BrakKomunikacji] := enumAlarmWartosc.StanNormalny;
	xBrakKomunikacjiEnOcean := FALSE;
	arErrorKlasa[enumPPPSZadajnikError.BrakKomunikacji] := enumPPPSZadajnikErrorKlasa.BrakKomunikacji;
	IF xPoInicjalizacji THEN
		fnZapiszKomunikat(	sCalyKomunikat := '' ,
							sTypKomunikatu := 'E' ,
							sMnemonik := sMnemonik ,
							sMACAdres := sMACAdres ,
							sIDNadawcy := sIdInstancji ,
							sIDOdbiorcy := sIdAplikacji ,
							sDaneZapasowe := sDaneZapasowe ,
							sDane := fnKomunikatDaneError(xAktywny := FALSE , intKlasa := enumPPPSZadajnikErrorKlasa.BrakKomunikacji , intNumer := enumPPPSZadajnikError.BrakKomunikacji),
							arTablicaKomunikatow := arTablicaKomunikatow ,
							intTablicaKomunikatowZnacznikZapisu := intTablicaKomunikatowZnacznikZapisu ,
							intTablicaKomunikatowRozmiar := intTablicaKomunikatowRozmiar ,
							sWyslanyKomunikat := sWyslanyKomunikatDummy);
	END_IF
END_IF
// Alarm czujnika temperatury
IF arErrorStan[enumPPPSZadajnikError.AlarmCzujnika] <> enumAlarmWartosc.StanAlarmowy AND xBladBrakZmianyTemperatury AND arModbusStatusKomunikacji[bAdres] = enumModbusStatus.KomunikacjaPrawidlowa THEN
	arErrorStan[enumPPPSZadajnikError.AlarmCzujnika] := enumAlarmWartosc.StanAlarmowy;
	arErrorKlasa[enumPPPSZadajnikError.AlarmCzujnika] := enumPPPSZadajnikErrorKlasa.AlarmCzujnika;
	IF xPoInicjalizacji THEN
		fnZapiszKomunikat(	sCalyKomunikat := '' ,
							sTypKomunikatu := 'E' ,
							sMnemonik := sMnemonik ,
							sMACAdres := sMACAdres ,
							sIDNadawcy := sIdInstancji ,
							sIDOdbiorcy := sIdAplikacji ,
							sDaneZapasowe := sDaneZapasowe ,
							sDane := fnKomunikatDaneError(xAktywny := TRUE , intKlasa := enumPPPSZadajnikErrorKlasa.AlarmCzujnika , intNumer := enumPPPSZadajnikError.AlarmCzujnika),
							arTablicaKomunikatow := arTablicaKomunikatow ,
							intTablicaKomunikatowZnacznikZapisu := intTablicaKomunikatowZnacznikZapisu ,
							intTablicaKomunikatowRozmiar := intTablicaKomunikatowRozmiar ,
							sWyslanyKomunikat := sWyslanyKomunikatDummy);
	END_IF
END_IF

IF arErrorStan[enumPPPSZadajnikError.AlarmCzujnika] <> enumAlarmWartosc.StanNormalny AND NOT xBladBrakZmianyTemperatury AND arModbusStatusKomunikacji[bAdres] = enumModbusStatus.KomunikacjaPrawidlowa THEN
	arErrorStan[enumPPPSZadajnikError.AlarmCzujnika] := enumAlarmWartosc.StanNormalny;
	arErrorKlasa[enumPPPSZadajnikError.AlarmCzujnika] := enumPPPSZadajnikErrorKlasa.AlarmCzujnika;
	IF xPoInicjalizacji THEN
		fnZapiszKomunikat(	sCalyKomunikat := '' ,
							sTypKomunikatu := 'E' ,
							sMnemonik := sMnemonik ,
							sMACAdres := sMACAdres ,
							sIDNadawcy := sIdInstancji ,
							sIDOdbiorcy := sIdAplikacji ,
							sDaneZapasowe := sDaneZapasowe ,
							sDane := fnKomunikatDaneError(xAktywny := FALSE , intKlasa := enumPPPSZadajnikErrorKlasa.AlarmCzujnika , intNumer := enumPPPSZadajnikError.AlarmCzujnika),
							arTablicaKomunikatow := arTablicaKomunikatow ,
							intTablicaKomunikatowZnacznikZapisu := intTablicaKomunikatowZnacznikZapisu ,
							intTablicaKomunikatowRozmiar := intTablicaKomunikatowRozmiar ,
							sWyslanyKomunikat := sWyslanyKomunikatDummy);
	END_IF
END_IF

// Plakietka pomieszczenia (numer piętra.numer pomieszczenia)
sPlakietkaHMI := CONCAT(STR1 := MID(sIdInstancji, LEN := 2, POS := 3), '.');
sPlakietkaHMI := CONCAT(sPlakietkaHMI, MID(STR := sIdInstancji, LEN := 3, POS := 7));
          
END_FUNCTION_BLOCK
